// TIA Portal V17 export
// export: Created 2023-05-07T12:12:09.5629725Z, ExportSetting WithDefaults, DisplayName Totally Integrated Automation Portal, DisplayVersion V17, DisplayName TIA Portal Openness, DisplayVersion V17, DisplayName TIA Portal Version Control Interface, DisplayVersion V17, DisplayName TIA Portal Test Suite Advanced, DisplayVersion V17, DisplayName STEP 7 Professional, DisplayVersion V17, DisplayName SIMATIC Energy Suite, DisplayVersion V17, DisplayName STEP 7 Safety, DisplayVersion V17, DisplayName WinCC Professional, DisplayVersion V17
FUNCTION "ValueAssignment" : Void   // FC9, LAD
TITLE = ValueAssignment
{ S7_Optimized_Access := 'TRUE' }
VERSION : 0.1
// stored: AutoNumber true, IsIECCheckEnabled false, SetENOAutomatically false, UDAEnableTagReadback false
BEGIN

REGION Network 1: Move: rate
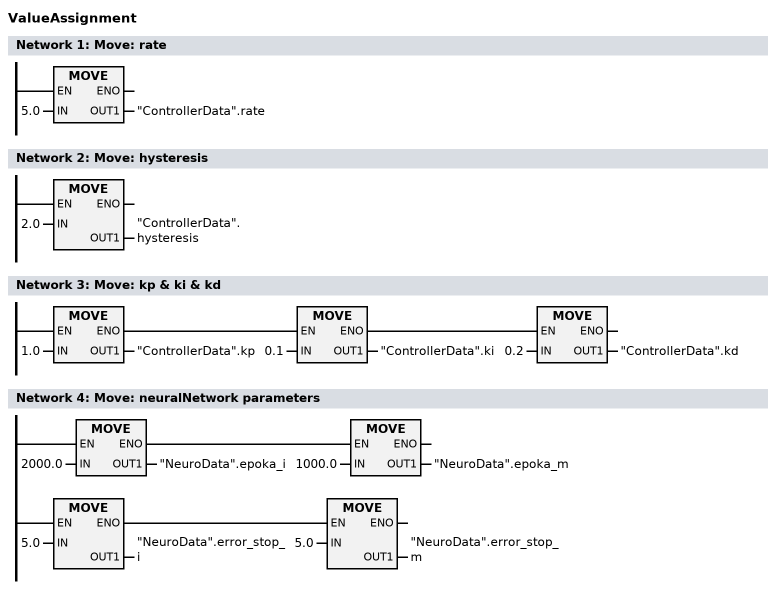
   RUNG wire#powerrail
      Move(in := 5.0, out1 => "ControllerData".rate)
   END_RUNG
   // the same network as SCL:
   "ControllerData".rate := 5.0;
END_REGION

REGION Network 2: Move: hysteresis
   RUNG wire#powerrail
      Move(in := 2.0, out1 => "ControllerData".hysteresis)
   END_RUNG
   // the same network as SCL:
   "ControllerData".hysteresis := 2.0;
END_REGION

REGION Network 3: Move: kp & ki & kd
   RUNG wire#powerrail
      Move(in := 1.0, out1 => "ControllerData".kp)
      Move(in := 0.1, out1 => "ControllerData".ki)
      Move(in := 0.2, out1 => "ControllerData".kd)
   END_RUNG
   // the same network as SCL:
   "ControllerData".kp := 1.0;
   "ControllerData".ki := 0.1;
   "ControllerData".kd := 0.2;
END_REGION

REGION Network 4: Move: neuralNetwork parameters
   RUNG wire#powerrail
      Move(in := 2000.0, out1 => "NeuroData".epoka_i)
      Move(in := 1000.0, out1 => "NeuroData".epoka_m)
   END_RUNG
   RUNG wire#powerrail
      Move(in := 5.0, out1 => "NeuroData".error_stop_i)
      Move(in := 5.0, out1 => "NeuroData".error_stop_m)
   END_RUNG
   // the same network as SCL:
   "NeuroData".epoka_i := 2000.0;
   "NeuroData".epoka_m := 1000.0;
   "NeuroData".error_stop_i := 5.0;
   "NeuroData".error_stop_m := 5.0;
END_REGION
END_FUNCTION
